FUNCTION A_TIME : ST_Arg
VAR_INPUT
	obj	: REFERENCE TO TIME;
END_VAR

IF __ISVALIDREF(obj) THEN
	A_TIME.eType := E_ArgType.TimeArg;
	A_TIME.pData := ADR(obj);
	A_TIME.nSize := SIZEOF(TIME);
END_IF

END_FUNCTION

(* stored: Version 1.1.0.1, ProductVersion 3.1.4024.15
   POU A_TIME: Id {9e666b4c-d7c0-48d2-bd36-5d6a42be3d47}, SpecialFunc None *)
